// TIA Portal V18 export
FUNCTION "FC_AI" : Void   // FC9, STL
{ S7_Optimized_Access := 'TRUE' }
VERSION : 0.1
// stored: AutoNumber true, UDAEnableTagReadback false
BEGIN

NETWORK
TITLE = 


      CALL  "FC_AnalogInCoverter"
      ( in_AnalogData  := "ina_InductiveResult",
        in_ScaleMax    := 5.0,
        in_SacaleMin   := 0.0,
        out_AnalogData := "DB_AI".ina_InductiveResult
      );

      CALL  "FC_AnalogInCoverter"
      ( in_AnalogData  := "ina_1",
        in_ScaleMax    := 0.0,
        in_SacaleMin   := 0.0,
        out_AnalogData := "DB_AI".ina_1
      );

      CALL  "FC_AnalogInCoverter"
      ( in_AnalogData  := "in_BaseAxis",
        in_ScaleMax    := 180.0,
        in_SacaleMin   := -180.0,
        out_AnalogData := "DB_AI".ina_BaseAxis
      );

      CALL  "FC_AnalogInCoverter"
      ( in_AnalogData  := "ina_Arm1Axis",
        in_ScaleMax    := 180.0,
        in_SacaleMin   := -180.0,
        out_AnalogData := "DB_AI".ina_Arm1Axis
      );

      CALL  "FC_AnalogInCoverter"
      ( in_AnalogData  := "ina_Arm2Axis",
        in_ScaleMax    := 180.0,
        in_SacaleMin   := -180.0,
        out_AnalogData := "DB_AI".ina_Arm2Axis
      );

      CALL  "FC_AnalogInCoverter"
      ( in_AnalogData  := "ina_Arm3Axis",
        in_ScaleMax    := 180.0,
        in_SacaleMin   := -180.0,
        out_AnalogData := "DB_AI".ina_Arm3Axis
      );


      CALL  "FC_AnalogInCoverter"
      ( in_AnalogData  := "ina_ToolAxis",
        in_ScaleMax    := 180.0,
        in_SacaleMin   := -180.0,
        out_AnalogData := "DB_AI".ina_ToolAxis
      );

      CALL  "FC_AnalogInCoverter"
      ( in_AnalogData  := "ina_7",
        in_ScaleMax    := 0.0,
        in_SacaleMin   := 0.0,
        out_AnalogData := "DB_AI".ina_7
      );

      CALL  "FC_AnalogInCoverter"
      ( in_AnalogData  := "ina_8",
        in_ScaleMax    := 0.0,
        in_SacaleMin   := 0.0,
        out_AnalogData := "DB_AI".ina_8
      );

      CALL  "FC_AnalogInCoverter"
      ( in_AnalogData  := "ina_9",
        in_ScaleMax    := 0.0,
        in_SacaleMin   := 0.0,
        out_AnalogData := "DB_AI".ina_9
      );

      CALL  "FC_AnalogInCoverter"
      ( in_AnalogData  := "ina_HorizontalAxis",
        in_ScaleMax    := 9.5,
        in_SacaleMin   := 0.0,
        out_AnalogData := "DB_AI".ina_HorizontalAxis
      );

      CALL  "FC_AnalogInCoverter"
      ( in_AnalogData  := "ina_VerticalAxis",
        in_ScaleMax    := 5.0,
        in_SacaleMin   := 0.0,
        out_AnalogData := "DB_AI".ina_VerticalAxis
      );




END_FUNCTION
